// TIA Portal V20 export
TYPE "LConSMC_typeWinderConfig"
// Konfigurationsdaten des Wicklers / Configuration data of the winder
// stored: Access Published
   STRUCT
      positionControlled : Bool := FALSE;   // TRUE: Enable MoveVelocity position controlled in case of positioning axis
      axisCtrl : Bool := TRUE;   // FALSE: Setpoints (Velocity, Torque) are not forwarded to the axis. An external axis control must be realized (see diagnostic outputs "referenceVelocity" and "diameterFactor") TRUE: Setpoints (Velocity, Torque) are forwarded to the axis internally
      jogVelocity : Real := 0.0;   // [m/min oder ft/min] Web velocity to jog the drive via the inputs "jogPos" and "jogNeg"
      overrideVelocity : Real := 0.0;   // [m/min or ft/min] Additive velocity offset for speed controller This value is only needed for the torque controlled modes (controlMode = 1-3)
      maxVelocity : Real := 0.0;   // [m/min or ft/min] Maximum possible web velocity. Maximum speed setpoint of the axis is limited to maxVelocity (+ overrideVelocity) and minimum diameter
      getAxisConfigAtStart : Bool := TRUE;   // TRUE: Readout gear,reference torque and units from axis with rising edge. FALSE: Take config values
      noOfSamplesLineVelocity : UInt := 1;   // Number of samples for moving average filter of line velocity setpoint for synchronizing to a moving web
      unitConfiguration { S7_SetPoint := 'True'} : "LConSMC_typeUnitConfiguration";   // Configuration of the units
      winderDynamics { S7_SetPoint := 'True'} : "LConSMC_typeAxisDynamics";   // Configuration of the axis dynamics
      torquePrecontrolConfig { S7_SetPoint := 'True'} : "LConSMC_typeTorquePrecontrolConfig";   // Configuration parameters for torque precontrol
      diamConfig { S7_SetPoint := 'True'} : "LConSMC_typeDiamConfig";   // Configuration parameters for diameter calculation
      technologyControllerConfig { S7_SetPoint := 'True'} : "LConSMC_typeTechnologyControllerConfig";   // Configuration parameters for technology controller (Dancer or load cell)
      webbreakDetectionConfig { S7_SetPoint := 'True'} : "LConSMC_typeWebbreakDetectConfig";   // Configuration parameters for webbreak detection
   END_STRUCT;
END_TYPE
